FUNCTION_BLOCK Calibracion_Po_calc
VAR_INPUT
	Dosis:REAL;
	Tinyeccion:DINT;
	PesoBatch:REAL;
	Tolerancia:REAL;
	Pausa:BOOL;
	PesoMaxConte:REAL;
	PesoConte:REAL;
END_VAR
VAR_OUTPUT
	Error:REAL;
	Peso_en_contenedor:REAL;
	PesoCalibra:REAL;
	PesoProm:REAL;
    Muestra2:BOOL;
END_VAR
VAR_IN_OUT
	Inicio:BOOL;
	Coef:REAL;
	Inyectar:BOOL;
	Tarar:BOOL;
	CantPesadas:INT;
	ContLleno:BOOL;
	Finalizado:BOOL;	
END_VAR
VAR

	IniciarCal: R_TRIG;
	Caudal:REAL;
	PesoMax:REAL;
	PesoMin:REAL;
	Calibrando:BOOL;
	IniInyectar:R_TRIG;
	FinInyectar:F_TRIG;
	Inyectando:BOOL;
	PesoIni:REAL;
	Pesada:ARRAY [1..6]OF REAL;
	Muestra1:BOOL;
	PromMuestra:REAL;
	IniCal:BOOL;
	IniIny:BOOL;
	FinIny:BOOL;
	tDemoraFinIny:TON;
	tDemoraFinIny2:TON;
	StepCal:INT;
	bContenedorLleno:F_TRIG;
	borrarContenedorLleno:BOOL;
	CancelarCal:F_TRIG;
	CanCal: BOOL;
	Teste: INT;
	i: INT;
	PromMuestra2: REAL;
END_VAR


IniciarCal(CLK:=Inicio , Q=>IniCal );
IF IniCal THEN
	StepCal:=1;
	IniCal:=0;
END_IF
CancelarCal(CLK:=Inicio , Q=>CanCal );

IF CanCal  THEN
	StepCal:=0;
	Pausa:=FALSE;
	CantPesadas:=0;
	Calibrando:=FALSE;
	Muestra1:=FALSE;
	Muestra2:=FALSE;
	CanCal:=0;
END_IF
PesoCalibra:=Dosis*PesoBatch/100;
bContenedorLleno(CLK:=ContLleno ,Q=>borrarContenedorLleno );
IF borrarContenedorLleno THEN
	Peso_en_contenedor:=0;
	Tarar:=TRUE;
	borrarContenedorLleno:=0;
END_IF

CASE StepCal OF
	1: 
		IF Tinyeccion=0 THEN
			Tinyeccion:=1;
		END_IF
		Tarar:=TRUE;
		Caudal:=PesoCalibra/DINT_TO_REAL (Tinyeccion);
		PesoMax:=(PesoCalibra*(1+Tolerancia/100))/1000;
		PesoMin:=(PesoCalibra*(1-Tolerancia/100))/1000;
		Pesada[1]:=0;
		Pesada[2]:=0;
		Pesada[3]:=0;
		Pesada[4]:=0;
		Pesada[5]:=0;
		Pesada[6]:=0;
		Finalizado:=0;
		Peso_en_contenedor:=0;
		CantPesadas:=0;
		Calibrando:=TRUE;
		IniCal:=0;
		StepCal:=2;
		
	2: 	Inyectar:=TRUE;
		Muestra1:=TRUE;
		//Tarar:=FALSE;
		PesoIni:=PesoConte;
		StepCal:=3;
		
	3: 	tDemoraFinIny(IN:=NOT Inyectar,PT:=T#10S);;
		IF tDemoraFinIny.Q THEN
			Tarar:=FALSE;
			StepCal:=4;
		END_IF
		
	4: 	CantPesadas := CantPesadas + 1;	
		Pesada[CantPesadas] := PesoConte - PesoIni;
		Peso_en_contenedor := Peso_en_contenedor + Pesada[CantPesadas];
		StepCal := 5;
		
	5:	IF Peso_en_contenedor > (0.9 * PesoMaxConte) THEN
			ContLleno:=1;
		ELSE
			StepCal:=6;		
		END_IF;
		
	6:		IF CantPesadas<3 THEN
				IF NOT Pausa THEN
					StepCal:=2;
				END_IF
			ELSE
				StepCal:=7;	
			END_IF;
	
	7://Calculo error muestra1
		IF CantPesadas=3 AND Muestra1 AND NOT Muestra2 AND NOT Inyectar THEN
			PromMuestra:=(Pesada[1]+Pesada[2]+Pesada[3])/3;
			IF (PromMuestra<=PesoMax) AND (PromMuestra>=PesoMin) THEN
				Muestra2:=TRUE;
				StepCal:=8;	
			ELSE
				//Coef:=Coef*	(PesoCalibra*0.001)/PromMuestra;
				
				IF PesoCalibra / (PromMuestra * 1000) >= 3 THEN
					Teste := 1;
					Coef := Coef + 0.4;
				ELSIF PesoCalibra / (PromMuestra * 1000) < 3 AND PesoCalibra / (PromMuestra * 1000) >= 2 THEN
					Teste := 2;
					Coef := Coef + 0.03;
				ELSIF PesoCalibra / (PromMuestra * 1000) < 2 AND PesoCalibra / (PromMuestra * 1000) >= 1 THEN
					Teste := 3;
					Coef := Coef + 0.03;
				ELSIF PesoCalibra / (PromMuestra * 1000) < 1 AND PesoCalibra / (PromMuestra * 1000) >= 0.5 THEN
					Teste := 4;
					Coef := Coef - 0.03;
				ELSE
					Coef := Coef - 0.1;
					Teste := 5;
				END_IF
				//Coef:=Coef+((((PesoCalibra*0.001)-PromMuestra)/(PesoCalibra*0.001))/1);
				Muestra1:=FALSE;
				CantPesadas:=0;	
				StepCal:=2;	
			FOR i := 1 TO 6 DO
				Pesada[i] := 0;
			END_FOR		
			END_IF		
		END_IF;
		
	8:	Inyectar:=TRUE;
		PesoIni:=PesoConte;
		StepCal:=9;
		
	9:	tDemoraFinIny2(IN:=NOT Inyectar,PT:=T#10S);;
		IF tDemoraFinIny2.Q THEN
			StepCal:=10;
		END_IF;
		
	10:	CantPesadas:=CantPesadas+1;	
		Pesada[CantPesadas]:=PesoConte-PesoIni;
		Peso_en_contenedor:=Peso_en_contenedor+Pesada[CantPesadas];
		StepCal:=11;
		
	11:	IF Peso_en_contenedor>(0.9*PesoMaxConte) THEN
			ContLleno:=1;
		ELSE
			StepCal:=12;		
		END_IF;
			
	12:		IF CantPesadas<6 THEN
				IF NOT Pausa THEN
					StepCal:=8;
				END_IF	
			ELSE
				StepCal:=13;	
			END_IF;
	
	13:	
			PromMuestra2:=(Pesada[4]+Pesada[5]+Pesada[6])/3;
		IF ((PromMuestra2<PesoMax) AND (PromMuestra2>PesoMin)) THEN
			PesoProm:=((Pesada[1]+Pesada[2]+Pesada[3]+Pesada[4]+Pesada[5]+Pesada[6])/6)*1000;
			Error:=((PesoCalibra-PesoProm)/PesoCalibra)*100;
			Inicio:=FALSE;
			Muestra1:=FALSE;
			Muestra2:=FALSE;
			Calibrando:=FALSE;
			Finalizado:=TRUE;
			Tarar:=0;
			StepCal:=0;	
		ELSE
			//Coef:=Coef+((((PesoCalibra*0.001)-PromMuestra)/(PesoCalibra*0.001))/100);
			//Coef:=Coef*(PesoCalibra*0.001)/PromMuestra;
			IF PesoCalibra / (PromMuestra * 1000) >= 3 THEN
				Coef := Coef + 0.4;
			ELSIF PesoCalibra / (PromMuestra * 1000) < 3 AND PesoCalibra / (PromMuestra * 1000) >= 2 THEN
				Coef := Coef + 0.03;
			ELSIF PesoCalibra / (PromMuestra * 1000) < 2 AND PesoCalibra / (PromMuestra * 1000) >= 1 THEN
				Coef := Coef + 0.03;
			ELSIF PesoCalibra / (PromMuestra * 1000) < 1 AND PesoCalibra / (PromMuestra * 1000) >= 0.5 THEN
				Coef := Coef - 0.03;
			ELSE
				Coef := Coef - 0.1;
			END_IF
			Muestra1:=FALSE;
			Muestra2:=FALSE;
			CantPesadas:=0;
			StepCal:=2;	
			FOR i := 1 TO 6 DO
				Pesada[i] := 0;
			END_FOR
		END_IF;		
		
END_CASE

//Faz a média de valores de acordo com a contagem de pesagens
IF CantPesadas > 0 THEN
	//PromMuestra:=(Pesada[1]+Pesada[2]+Pesada[3]+Pesada[4]+Pesada[5]+Pesada[6])/CantPesadas;
	PromMuestra := 0;
	FOR i := 1 TO CantPesadas DO
		PromMuestra := PromMuestra + (Pesada[i]/CantPesadas);
	END_FOR
END_IF;

//Verifica se o recipiente está cheio
IF Peso_en_contenedor>(0.9*PesoMaxConte) THEN
	ContLleno:=1;
END_IF;

END_FUNCTION_BLOCK

(* stored: Version 1.1.0.1, ProductVersion 3.1.4024.14
   POU Calibracion_Po_calc: Id {7b335178-e7a5-4c39-a984-17c7504860f5}, SpecialFunc None *)
